TYPE ST_LAB_CaseData :
STRUCT
	aOuters		: ARRAY[1..50] OF ST_LAB_OuterData;
END_STRUCT
END_TYPE

(* stored: Version 1.1.0.1
   DUT ST_LAB_CaseData: Id {7b26a288-e3a8-4529-8e02-0e89e7ef32e4} *)
